FUNCTION Convert_DATE_TO_LWORD : BOOL
VAR_INPUT
	in : DATE;
	out : REFERENCE TO LWORD;
END_VAR
VAR
	converted : LWORD;
END_VAR

converted := DATE_TO_LWORD(in);

IF (LWORD_TO_DATE(converted) <> in) THEN
	RETURN;
END_IF

out := converted;
Convert_DATE_TO_LWORD := TRUE;

END_FUNCTION

(* stored: Version 1.1.0.1, ProductVersion 3.1.4024.12
   POU Convert_DATE_TO_LWORD: Id {0c857252-3c2b-46c2-bda8-720879c00352}, SpecialFunc None *)
